// TwinCAT 3 PLC project PlcIotHttpSamplesPhilipsHue
// ProgramVersion: 3.1.4023.0
// libraries:
//   Tc2_Standard, * (Beckhoff Automation GmbH)
//   Tc2_System, * (Beckhoff Automation GmbH)
//   Tc2_Utilities, * (Beckhoff Automation GmbH)
//   Tc3_IotBase, * (Beckhoff Automation GmbH)
//   Tc3_JsonXml, * (Beckhoff Automation GmbH)
//   Tc3_Module, * (Beckhoff Automation GmbH)
// project tree:
//   / PlcTask.TcTTO
//   POUs/ MAIN.TcPOU
//   POUs/Philips Hue/ FB_TestHTTP_Put_PhilipsHue.TcPOU
// (motion and I/O tree: see PLC project plciothttpsamplespostman)
// real-time tasks:
//   TASK PlcTask: cycle T#10ms, priority 20, ADS port 350
//   TASK PlcTask1: cycle T#10ms, priority 21, ADS port 351
//   TASK PlcTask2: cycle T#10ms, priority 22, ADS port 352
//   TASK PlcTask3: cycle T#10ms, priority 23, ADS port 353
//   TASK PlcTask4: cycle T#10ms, priority 24, ADS port 354
//   TASK PlcTask5: cycle T#10ms, priority 25, ADS port 355
//   TASK PlcTask6: cycle T#10ms, priority 26, ADS port 356

CONFIGURATION PlcIotHttpSamplesPhilipsHue
    RESOURCE PLC ON TwinCAT3
        TASK PlcTask(INTERVAL := T#10ms, PRIORITY := 24);
        PROGRAM MAIN WITH PlcTask : MAIN;
    END_RESOURCE
END_CONFIGURATION

// ---- POUs/MAIN.TcPOU
PROGRAM MAIN
VAR
	// trigger command execution for Philips Hue samples
	bPutPhilipsHue 					: BOOL;

	fbHttpClientPhilipsHue			: FB_IotHttpClient :=(sHostName:='172.17.38.83',
									bKeepAlive:=TRUE, tConnectionTimeout:=T#10S);

	fbHttpPutPhilipsHue				: FB_TestHTTP_Put_PhilipsHue;
	
	bBlinkingMode					: BOOL;
	fbTimer							: TON:=(PT:=T#500MS);
	nColor               			: UINT;
END_VAR

// init client parameters at startup
IF NOT fbHttpClientPhilipsHue.bConfigured THEN 
	fbHttpClientPhilipsHue.nHostPort:= 80;
	fbHttpClientPhilipsHue.stTLS.bNoServerCertCheck:=TRUE;
END_IF

IF fbHttpClientPhilipsHue.bConfigured THEN
	fbHttpPutPhilipsHue(bSend:=bPutPhilipsHue, fbClient:=fbHttpClientPhilipsHue, nColor:=nColor);
END_IF

IF bBlinkingMode THEN
	fbTimer(IN:=NOT fbTimer.Q);
	IF fbTimer.Q THEN
		nColor:=nColor+5000;
		IF nColor=65000 THEN
			nColor:=0;
		END_IF
		IF bPutPhilipsHue THEN
			bPutPhilipsHue:=FALSE;
		ELSE 
			bPutPhilipsHue:=TRUE;
		END_IF
	END_IF
END_IF

fbHttpClientPhilipsHue.Execute();

END_PROGRAM

// ---- POUs/Philips Hue/FB_TestHTTP_Put_PhilipsHue.TcPOU
FUNCTION_BLOCK FB_TestHTTP_Put_PhilipsHue
VAR_INPUT
	bSend				: BOOL;
	nColor				: UINT;
END_VAR
VAR_IN_OUT
	fbClient			: FB_IotHttpClient;
END_VAR
VAR_OUTPUT
	bBusy				: BOOL;
	bError				: BOOL;
END_VAR
VAR
	fbRequest			: FB_IotHttpRequest;
	fbJson				: FB_JsonDomParser;
	fbJsonWriter		: FB_JsonSaxWriter;
	nState				: UDINT;
	RisingEdge			: R_TRIG;
	
	bGetContentResult	: BOOL;
	sContent			: STRING(511);
	sSend				: STRING(511);
	
	bGetJsonResult		: BOOL;
	jsonDoc				: SJsonValue;
	jsonVal				: SJsonValue;
	sResultValue		: STRING;
	
	nReqCount			: UDINT;	
	nResCount			: UDINT;
	nValidResCount		: UDINT;
	nErrCount			: UDINT;
	
	fbTimer				: TON;
	bLightOn			: BOOL;
END_VAR

RisingEdge(CLK:= bSend );

CASE nState OF
0:	
		fbJsonWriter.StartObject();
		fbJsonWriter.AddKey('on');
		fbJsonWriter.AddBool(TRUE);
		fbJsonWriter.AddKey('sat');
		fbJsonWriter.AddUdint(50);
		fbJsonWriter.AddKey('bri');
		fbJsonWriter.AddUdint(100);
		fbJsonWriter.AddKey('hue');
		fbJsonWriter.AddUdint(nColor);
		fbJsonWriter.EndObject();
		sSend:=fbJsonWriter.GetDocument();
		fbJsonWriter.ResetDocument();
	IF RisingEdge.Q THEN 
		IF fbRequest.SendRequest(sUri:='/api/qiyut7ubQQQv2xKJfFe9cVvIroUGHtIk2eYsIfGX/lights/1/state', fbClient:=fbClient, eRequestType:=ETcIotHttpRequestType.HTTP_PUT, pContent:=ADR(sSend), nContentSize:=LEN2(ADR(sSend)), 0) THEN				
			nState:= 1;
			nReqCount:= nReqCount+1;
			bBusy:= TRUE;
			bError:= FALSE;
		END_IF					
	END_IF
1:
	IF NOT fbRequest.bBusy THEN
		bError:= TRUE;
		IF NOT fbRequest.bError THEN				 
			bGetContentResult:= fbRequest.GetContent(pContent:= ADR(sContent), nContentSize:= SIZEOF(sContent), bSetNullTermination:= TRUE);
			IF fbRequest.nStatusCode >= 200 AND fbRequest.nStatusCode < 300 THEN
				bGetJsonResult:= FALSE;
				jsonDoc:= fbRequest.GetJsonDomContent(fbJson);
				IF jsonDoc <> 0 THEN
					; // do something with status response
					nValidResCount:= nValidResCount+1;
					bError:= FALSE;	
				END_IF							
				nResCount:= nResCount+1;			
			END_IF
		END_IF
		nState:= 0;
		bBusy:= FALSE;
		IF bError THEN
			nErrCount:= nErrCount+1;
		END_IF
	END_IF  	
END_CASE

END_FUNCTION_BLOCK
